// TIA Portal V20 export
TYPE "LBP_typeModularMcpAxisInput"
TITLE = Modular MCP image / Image MCP modulaire
// Input image of axis keypad for modular MCP / Image des entrées du champ de touches d'axe pour MCP modulaires
   STRUCT
      minus : Bool;   // input image n+0 bit 0 / Image des entrées n+0 bit 0
      rapidTraverse : Bool;   // input image n+0 bit 1 / Image des entrées n+0 bit 1
      plus : Bool;   // input image n+0 bit 2 / Image des entrées n+0 bit 2
      key3 : Bool;   // input image n+0 bit 3 / Image des entrées n+0 bit 3
      tcs : Bool;   // input image n+0 bit 4 / Image des entrées n+0 bit 4
      mcsWcs : Bool;   // input image n+0 bit 5 / Image des entrées n+0 bit 5
      key6 : Bool;   // input image n+0 bit 6 / Image des entrées n+0 bit 6
      key7 : Bool;   // input image n+0 bit 7 / Image des entrées n+0 bit 7
      key8 : Bool;   // input image n+1 bit 0 / Image des entrées n+1 bit 0
      axis4 : Bool;   // input image n+1 bit 1 / Image des entrées n+1 bit 1
      axis5 : Bool;   // input image n+1 bit 2 / Image des entrées n+1 bit 2
      axis6 : Bool;   // input image n+1 bit 3 / Image des entrées n+1 bit 3
      axisX : Bool;   // input image n+1 bit 4 / Image des entrées n+1 bit 4
      axisY : Bool;   // input image n+1 bit 5 / Image des entrées n+1 bit 5
      axisZ : Bool;   // input image n+1 bit 6 / Image des entrées n+1 bit 6
      reserved17 : Bool;
      feedrateStop : Bool;   // input image n+2 bit 0 / Image des entrées n+2 bit 0
      feedrateStart : Bool;   // input image n+2 bit 1 / Image des entrées n+2 bit 1
      key18 : Bool;   // input image n+2 bit 2 / Image des entrées n+2 bit 2
      reserved23 : Bool;
      reserved24 : Bool;
      reserved25 : Bool;
      reserved26 : Bool;
      reserved27 : Bool;
      spindleStop : Bool;   // input image n+3 bit 0 / Image des entrées n+3 bit 0
      spindleStart : Bool;   // input image n+3 bit 1 / Image des entrées n+3 bit 1
      key26 : Bool;   // input image n+3 bit 2 / Image des entrées n+3 bit 2
      reserved33 : Bool;
      reserved34 : Bool;
      reserved35 : Bool;
      reserved36 : Bool;
      reserved37 : Bool;
   END_STRUCT;
END_TYPE
